// TIA Portal V15.1 export
// export: Created 2024-06-21T08:41:15.0924027Z, ExportSetting WithDefaults, DisplayName Totally Integrated Automation Portal, DisplayVersion V15.1 Update 5, DisplayName TIA Portal Openness, DisplayVersion V15.1 Update 5, DisplayName SINAMICS Startdrive Advanced, DisplayVersion V15.1, DisplayName G130, G150, S120, S150, SINAMICS MV, S210, DisplayVersion V15.1, DisplayName G110M, G120, G120C, G120D, G120P, DisplayVersion V15.1, DisplayName STEP 7 Professional, DisplayVersion V15.1 Update 5, DisplayName STEP 7 Safety, DisplayVersion V15.1, DisplayName WinCC Professional, DisplayVersion V15.1 Update 5, DisplayName SIMATIC Visualization Architect, DisplayVersion V15.1
FUNCTION_BLOCK "LGBChain2W1S-MoviFitFCPN"   // FB6710, FBD
TITLE = LGBChain2W1S-C / LGBChain2W1S-MoviFitFCPN
{ S7_Optimized_Access := 'TRUE' }
VERSION : 0.1
// stored: AutoNumber false, IsIECCheckEnabled false, IsRetainMemResEnabled false, MemoryReserve 100, SetENOAutomatically False, UDAEnableTagReadback false
   VAR_INPUT
      I_ExitDet { ExternalAccessible := 'False'; ExternalVisible := 'False'; ExternalWritable := 'False'} : Bool;   // Stop Detection set
      I_EntranceDet { ExternalAccessible := 'False'; ExternalVisible := 'False'; ExternalWritable := 'False'} : Bool;   // Stop Detection Reset
      I_StopDetPrev { ExternalAccessible := 'False'; ExternalVisible := 'False'; ExternalWritable := 'False'} : Bool;   // Stop Detection previous conveyor
      I_SlipControlDet { ExternalAccessible := 'False'; ExternalVisible := 'False'; ExternalWritable := 'False'} : Bool;   // Slack Chain detection
      I_TrfInSetBegin { ExternalAccessible := 'False'; ExternalVisible := 'False'; ExternalWritable := 'False'} : Bool;   // Load Begin: condition to start transfer IN set
      I_TrfInSetIntlkOk { ExternalAccessible := 'False'; ExternalVisible := 'False'; ExternalWritable := 'False'} : Bool;   // Transfer IN Interlock Set OK
      I_TrfOutSetBegin { ExternalAccessible := 'False'; ExternalVisible := 'False'; ExternalWritable := 'False'} : Bool;   // Unload Begin: condition to start transfer OUT set
      I_TrfOutSetIntlkOk { ExternalAccessible := 'False'; ExternalVisible := 'False'; ExternalWritable := 'False'} : Bool;   // Transfer Out Interlock Set OK
      I_TrfInSetRdyDlv { ExternalAccessible := 'False'; ExternalVisible := 'False'; ExternalWritable := 'False'} : Bool;   // Ready to deliver: Signal from previous object set
      I_TrfInSetTM { ExternalAccessible := 'False'; ExternalVisible := 'False'; ExternalWritable := 'False'} : Bool;   // Transfer busy signal from previous equipement set
      I_TrfOutSetRdyRcv { ExternalAccessible := 'False'; ExternalVisible := 'False'; ExternalWritable := 'False'} : Bool;   // Ready to Receive: Signal from next object set
      I_TrfOutSetArrived { ExternalAccessible := 'False'; ExternalVisible := 'False'; ExternalWritable := 'False'} : Bool;   // Body Arrived: Signal from next object Set
      I_PBSet { ExternalAccessible := 'False'; ExternalVisible := 'False'; ExternalWritable := 'False'} : Bool;   // Push button for manual movement (on local panel) set
      I_PBReset { ExternalAccessible := 'False'; ExternalVisible := 'False'; ExternalWritable := 'False'} : Bool;   // Push button for manual movement (on local panel) Reset
      I_ManInfeedAllowedSet { ExternalAccessible := 'False'; ExternalVisible := 'False'; ExternalWritable := 'False'} : Bool;   // Manual Infeed Allowed Set (without PushButton)
      I_ManInfeedAllowedRes { ExternalAccessible := 'False'; ExternalVisible := 'False'; ExternalWritable := 'False'} : Bool;   // Manual Infeed Allowed Reset (without PushButton)
      I_MotorProtection { ExternalAccessible := 'False'; ExternalVisible := 'False'; ExternalWritable := 'False'} : Bool;   // Motorprotection
      I_ReleaseBrake { ExternalAccessible := 'False'; ExternalVisible := 'False'; ExternalWritable := 'False'} : Bool;   // Release brake
      I_SafetyOk { ExternalAccessible := 'False'; ExternalVisible := 'False'; ExternalWritable := 'False'} : Bool;   // Safety Ok
      I_MotionStopOk { ExternalAccessible := 'False'; ExternalVisible := 'False'; ExternalWritable := 'False'} : Bool;   // Safety Ok / The motion stop is Ok
      I_ProductionStop { ExternalAccessible := 'False'; ExternalVisible := 'False'; ExternalWritable := 'False'} : Bool;   // Production Stop
      I_ExtStartConveyor { ExternalAccessible := 'False'; ExternalVisible := 'False'; ExternalWritable := 'False'} : Bool;   // External Start Conveyor
      I_ChainEmptyTime { ExternalAccessible := 'False'; ExternalVisible := 'False'; ExternalWritable := 'False'} : DInt;   // Time to empty Chain (Msec)
      I_Speed { ExternalAccessible := 'False'; ExternalVisible := 'False'; ExternalWritable := 'False'} : Real;   // High speed Value (set-up %) / Speed Value (set-up %)
      I_SafetyStatusWord { ExternalAccessible := 'False'; ExternalVisible := 'False'; ExternalWritable := 'False'} : Word;   // Safety Status
      I_SafetyControlWord { ExternalAccessible := 'False'; ExternalVisible := 'False'; ExternalWritable := 'False'} : Word;   // Safety Control Word
   END_VAR
   VAR_OUTPUT
      O_ReleaseBrake { ExternalAccessible := 'False'; ExternalVisible := 'False'; ExternalWritable := 'False'} : Bool;   // Release the brake of the Motor
      O_Active { ExternalAccessible := 'False'; ExternalVisible := 'False'; ExternalWritable := 'False'} : Bool;   // Chain is Active
      O_TrfInSetRdyRcv { ExternalAccessible := 'False'; ExternalVisible := 'False'; ExternalWritable := 'False'} : Bool;   // Ready to Receive: Signal to previous object set
      O_TrfInSetArrived { ExternalAccessible := 'False'; ExternalVisible := 'False'; ExternalWritable := 'False'} : Bool;   // Body Arrived: Signal to previous object Set
      O_TrfOutSetRdyDlv { ExternalAccessible := 'False'; ExternalVisible := 'False'; ExternalWritable := 'False'} : Bool;   // Ready to Deliver: Signal to next object set
      O_TrfOutSetTM { ExternalAccessible := 'False'; ExternalVisible := 'False'; ExternalWritable := 'False'} : Bool;   // Transfer: Signal to next object set
      O_TrfInSetActive { ExternalAccessible := 'False'; ExternalVisible := 'False'; ExternalWritable := 'False'} : Bool;   // Transfer in set active
      O_TrfInSetFinished { ExternalAccessible := 'False'; ExternalVisible := 'False'; ExternalWritable := 'False'} : Bool;   // Transfer in set finished
      O_TrfOutSetActive { ExternalAccessible := 'False'; ExternalVisible := 'False'; ExternalWritable := 'False'} : Bool;   // Transfer out set active
      O_TrfOutSetFinished { ExternalAccessible := 'False'; ExternalVisible := 'False'; ExternalWritable := 'False'} : Bool;   // Transfer out set finished
      O_LedRoller { ExternalAccessible := 'False'; ExternalVisible := 'False'; ExternalWritable := 'False'} : Bool;   // Led of Chain
      O_AlarmABCondition { ExternalAccessible := 'False'; ExternalVisible := 'False'; ExternalWritable := 'False'} : Bool;   // Alarm AB Condition
      O_AlarmA { ExternalAccessible := 'False'; ExternalVisible := 'False'; ExternalWritable := 'False'} : Bool;   // Alarm A
      O_AlarmB { ExternalAccessible := 'False'; ExternalVisible := 'False'; ExternalWritable := 'False'} : Bool;   // Alarm B
      O_AlarmC { ExternalAccessible := 'False'; ExternalVisible := 'False'; ExternalWritable := 'False'} : Bool;   // Alarm C
      O_AlarmD { ExternalAccessible := 'False'; ExternalVisible := 'False'; ExternalWritable := 'False'} : Bool;   // Alarm D
      O_Occupied { ExternalAccessible := 'False'; ExternalVisible := 'False'; ExternalWritable := 'False'} : Bool;   // Chain Occupied
      H_AlarmDWord { ExternalAccessible := 'False'; ExternalVisible := 'False'; ExternalWritable := 'False'} : DWord;   // HMI Animation
   END_VAR
   VAR_IN_OUT
      IO_Modes : "Modes";   // Modes
      H_HMI : "H_HMI";   // Animation
      "H_GBChain2W1S-MoviFitFCPN" : "H_GBChain2W1S-MoviFitFCPN";   // Animation
      C_Config : "RollerConvMoviFitFCPNConfig";   // Config
   END_VAR
   VAR
      H_FncSelInHMI { ExternalAccessible := 'False'; ExternalVisible := 'False'; ExternalWritable := 'False'} : Bool;
      _SlipControl { ExternalAccessible := 'False'; ExternalVisible := 'False'; ExternalWritable := 'False'} : "L1AlarmMultiIn";   // FB
      _InitSlipControlCnt { ExternalAccessible := 'False'; ExternalVisible := 'False'; ExternalWritable := 'False'} : "LChangeOfState";   // FB
      AB_SlipControlAlm { ExternalAccessible := 'False'; ExternalVisible := 'False'; ExternalWritable := 'False'} : Bool;   // Alarm Slack Chain
      AC_TrfOutSetOverTime { ExternalAccessible := 'False'; ExternalVisible := 'False'; ExternalWritable := 'False'} : Bool;   // Timeout Transport Out Set
      AD_TrfOutSetInterlock { ExternalAccessible := 'False'; ExternalVisible := 'False'; ExternalWritable := 'False'} : Bool;   // Interlock Not Ok Transport Out Set
      AD_TrfInSetInterlock { ExternalAccessible := 'False'; ExternalVisible := 'False'; ExternalWritable := 'False'} : Bool;   // Interlock Not Ok Transport In Set
      AA_MotorProtector { ExternalAccessible := 'False'; ExternalVisible := 'False'; ExternalWritable := 'False'} : Bool;   // Motor Protection Tripped / Motorprotection Tripped
      AA_SafetySwitch { ExternalAccessible := 'False'; ExternalVisible := 'False'; ExternalWritable := 'False'} : Bool;   // Safety Switch Not Ok
      AB_STO { ExternalAccessible := 'False'; ExternalVisible := 'False'; ExternalWritable := 'False'} : Bool;   // Safety Switch Not Ok / Safety output to drive is active but no response from drive that the safety is ok
      AD_Warning { ExternalAccessible := 'False'; ExternalVisible := 'False'; ExternalWritable := 'False'} : Bool;   // Frequency Control
      AA_NoBusControl { ExternalAccessible := 'False'; ExternalVisible := 'False'; ExternalWritable := 'False'} : Bool;   // Frequency Control / Bus control inactive / Frekvensstyrning
      AB_Alarm { ExternalAccessible := 'False'; ExternalVisible := 'False'; ExternalWritable := 'False'} : Bool;   // Frequency Control
      AD_MotionStop { ExternalAccessible := 'False'; ExternalVisible := 'False'; ExternalWritable := 'False'} : Bool;   // Motion Stop
      AC_ConfigCalibrationAlm { ExternalAccessible := 'False'; ExternalVisible := 'False'; ExternalWritable := 'False'} : Bool;   // The Config values for Alarm Transfer time must be ALL zero or ALL different from zero
      AD_CalibrationSetWarn { ExternalAccessible := 'False'; ExternalVisible := 'False'; ExternalWritable := 'False'} : Bool;   // No High speed selected so Calibration is not possible for SET direction
      AC_ConfigRampAlm { ExternalAccessible := 'False'; ExternalVisible := 'False'; ExternalWritable := 'False'} : Bool;   // The config value for the ramp is not correct, must be zero or the config values for the calculation of the ramp must be ALL zero
      AC_ConfigRampCalcAlm { ExternalAccessible := 'False'; ExternalVisible := 'False'; ExternalWritable := 'False'} : Bool;   // The config values for the calculation of the ramp must be ALL different from zero
      PODataNotEnabled { ExternalAccessible := 'False'; ExternalVisible := 'False'; ExternalWritable := 'False'} : Bool;   // Bus control inactive
      SafetyOk { ExternalAccessible := 'False'; ExternalVisible := 'False'; ExternalWritable := 'False'} : Bool;   // Safety Ok
      SlipControlCond { ExternalAccessible := 'False'; ExternalVisible := 'False'; ExternalWritable := 'False'} : Bool;   // Alarm Slack Chain
      MotorLoopActive { ExternalAccessible := 'False'; ExternalVisible := 'False'; ExternalWritable := 'False'} : Bool;   // Motor Loop Active
      TrfInfeedHoldSet { ExternalAccessible := 'False'; ExternalVisible := 'False'; ExternalWritable := 'False'} : Bool;   // Transfer infeed hold set direction
      TrfOutSetCmd { ExternalAccessible := 'False'; ExternalVisible := 'False'; ExternalWritable := 'False'} : Bool;   // Command after Interlock to Motor set
      TrfOutfeedHoldSet { ExternalAccessible := 'False'; ExternalVisible := 'False'; ExternalWritable := 'False'} : Bool;   // Transfer outfeed hold set direction
      TrfInSetCmd { ExternalAccessible := 'False'; ExternalVisible := 'False'; ExternalWritable := 'False'} : Bool;   // Command after Interlock to Motor set
      MotorCmdSet { ExternalAccessible := 'False'; ExternalVisible := 'False'; ExternalWritable := 'False'} : Bool;   // Command to Motorloop High Speed Set
      MotorCmdRes { ExternalAccessible := 'False'; ExternalVisible := 'False'; ExternalWritable := 'False'} : Bool;   // Command to Motorloop High Speed Reset
      TrfInSetActive { ExternalAccessible := 'False'; ExternalVisible := 'False'; ExternalWritable := 'False'} : Bool;   // Load: Active (set)
      TrfOutSetActive { ExternalAccessible := 'False'; ExternalVisible := 'False'; ExternalWritable := 'False'} : Bool;   // Unload: active (set)
      TrfOutSetFinished { ExternalAccessible := 'False'; ExternalVisible := 'False'; ExternalWritable := 'False'} : Bool;   // Unload: finished (set)
      AlarmA { ExternalAccessible := 'False'; ExternalVisible := 'False'; ExternalWritable := 'False'} : Bool;   // Alarm A
      AlarmB { ExternalAccessible := 'False'; ExternalVisible := 'False'; ExternalWritable := 'False'} : Bool;   // Alarm B
      AlarmC { ExternalAccessible := 'False'; ExternalVisible := 'False'; ExternalWritable := 'False'} : Bool;   // Alarm C
      AlarmD { ExternalAccessible := 'False'; ExternalVisible := 'False'; ExternalWritable := 'False'} : Bool;   // Alarm D
      TrfOutSetRdyDlv { ExternalAccessible := 'False'; ExternalVisible := 'False'; ExternalWritable := 'False'} : Bool;   // Ready to Deliver: Signal to next object set
      TrfOutSetTM { ExternalAccessible := 'False'; ExternalVisible := 'False'; ExternalWritable := 'False'} : Bool;   // Transfer : Signal transfer memory to next object set
      TrfInSetTrfOutSetTM { ExternalAccessible := 'False'; ExternalVisible := 'False'; ExternalWritable := 'False'} : Bool;   // Transfer memory set
      TrfInSetRdyRcv { ExternalAccessible := 'False'; ExternalVisible := 'False'; ExternalWritable := 'False'} : Bool;   // Ready to Receive: Signal to previous object set
      TrfInSetArrived { ExternalAccessible := 'False'; ExternalVisible := 'False'; ExternalWritable := 'False'} : Bool;   // Body Arrived: Signal to previous object Set
      TrfInSetFinished { ExternalAccessible := 'False'; ExternalVisible := 'False'; ExternalWritable := 'False'} : Bool;   // Body Arrived: Signal to TrfOut module set (Reset TrfOutCmd)
      StopTrfOutSetCmd { ExternalAccessible := 'False'; ExternalVisible := 'False'; ExternalWritable := 'False'} : Bool;   // Body Arrived: Signal to previous object Set
      MotorLoopAlmCond { ExternalAccessible := 'False'; ExternalVisible := 'False'; ExternalWritable := 'False'} : Bool;   // Motor loop Alarm condition
      TrfOutSetAlmCond { ExternalAccessible := 'False'; ExternalVisible := 'False'; ExternalWritable := 'False'} : Bool;   // TrfOut set Alarm condition
      ChainStop { ExternalAccessible := 'False'; ExternalVisible := 'False'; ExternalWritable := 'False'} : Bool;   // Chain stop Productions Stop
      DlvSaturation { ExternalAccessible := 'False'; ExternalVisible := 'False'; ExternalWritable := 'False'} : Bool;   // Saturation for the diliver tranfer
      AlarmABCondition { ExternalAccessible := 'False'; ExternalVisible := 'False'; ExternalWritable := 'False'} : Bool;   // Alarm AB Condition
   END_VAR
   VAR RETAIN
      ChainEmpty { ExternalAccessible := 'False'; ExternalVisible := 'False'; ExternalWritable := 'False'} : Bool;   // Chain is Empty
   END_VAR
   VAR
      ChainEmptyTime { ExternalAccessible := 'False'; ExternalVisible := 'False'; ExternalWritable := 'False'} : DInt;   // Time to empty Chain (Msec)
      SlipControlPulseCount { ExternalAccessible := 'False'; ExternalVisible := 'False'; ExternalWritable := 'False'} : DInt;   // Temp
      SlipControlPosEdge1 { ExternalAccessible := 'False'; ExternalVisible := 'False'; ExternalWritable := 'False'} : Bool;   // Pos Edge
      SlipControlPosEdge2 { ExternalAccessible := 'False'; ExternalVisible := 'False'; ExternalWritable := 'False'} : Bool;   // Pos Edge
      InitSlipControlCounter { ExternalAccessible := 'False'; ExternalVisible := 'False'; ExternalWritable := 'False'} : Bool;   // Init
      ReleaseBrake { ExternalAccessible := 'False'; ExternalVisible := 'False'; ExternalWritable := 'False'} : Bool;   // Release brake
      ReadyForOperation { ExternalAccessible := 'False'; ExternalVisible := 'False'; ExternalWritable := 'False'} : Bool;   // Ready for operation
      _LTrfInSet { ExternalAccessible := 'False'; ExternalVisible := 'False'; ExternalWritable := 'False'} : "LGBTrfIn";   // FB
      _LTrfOutSet { ExternalAccessible := 'False'; ExternalVisible := 'False'; ExternalWritable := 'False'} : "LGBTrfOut";   // FB
      _Motor { ExternalAccessible := 'False'; ExternalVisible := 'False'; ExternalWritable := 'False'} : "LGBMotor2W2S-MoviFitFCPN";
      _ChainSlipControl { ExternalAccessible := 'False'; ExternalVisible := 'False'; ExternalWritable := 'False'} : "L1AlarmMultiIn";
      _ChainEmptyTimer { ExternalAccessible := 'False'; ExternalVisible := 'False'; ExternalWritable := 'False'} : TON_TIME;
   END_VAR
   VAR_TEMP
      H_HMITrfInSet : "H_HMI";   // Temp
      H_HMITrfOutSet : "H_HMI";   // Temp
      H_HMIMotor : "H_HMI";   // Temp
   END_VAR
   VAR_TEMP   // added for the SCL form of the ladder/FBD networks
      _w1 : Bool;
      _w2 : Bool;
      _w3 : Bool;
      _w4 : Bool;
   END_VAR
BEGIN

NETWORK
TITLE = **** 1 - Inputs **** Init Slip Control Set Direction
// Init Belt Control Set And Reset Direction
      CALL  #_InitSlipControlCnt
      ( I_In     := #I_SlipControlDet,
        O_OutPut := #InitSlipControlCounter
      );
      NOP   0;

      A(;
      O     #InitSlipControlCounter;
      O;
      A     #IO_Modes.LMode.ManualMode;
      A     #IO_Modes.LMode.AlarmResetPB;
      );
      JCN   NCSet;
      L     0;
      T     #SlipControlPulseCount;
NCSet:NOP   0;


REGION Network 2: **** 1 - Inputs **** Safety Ok
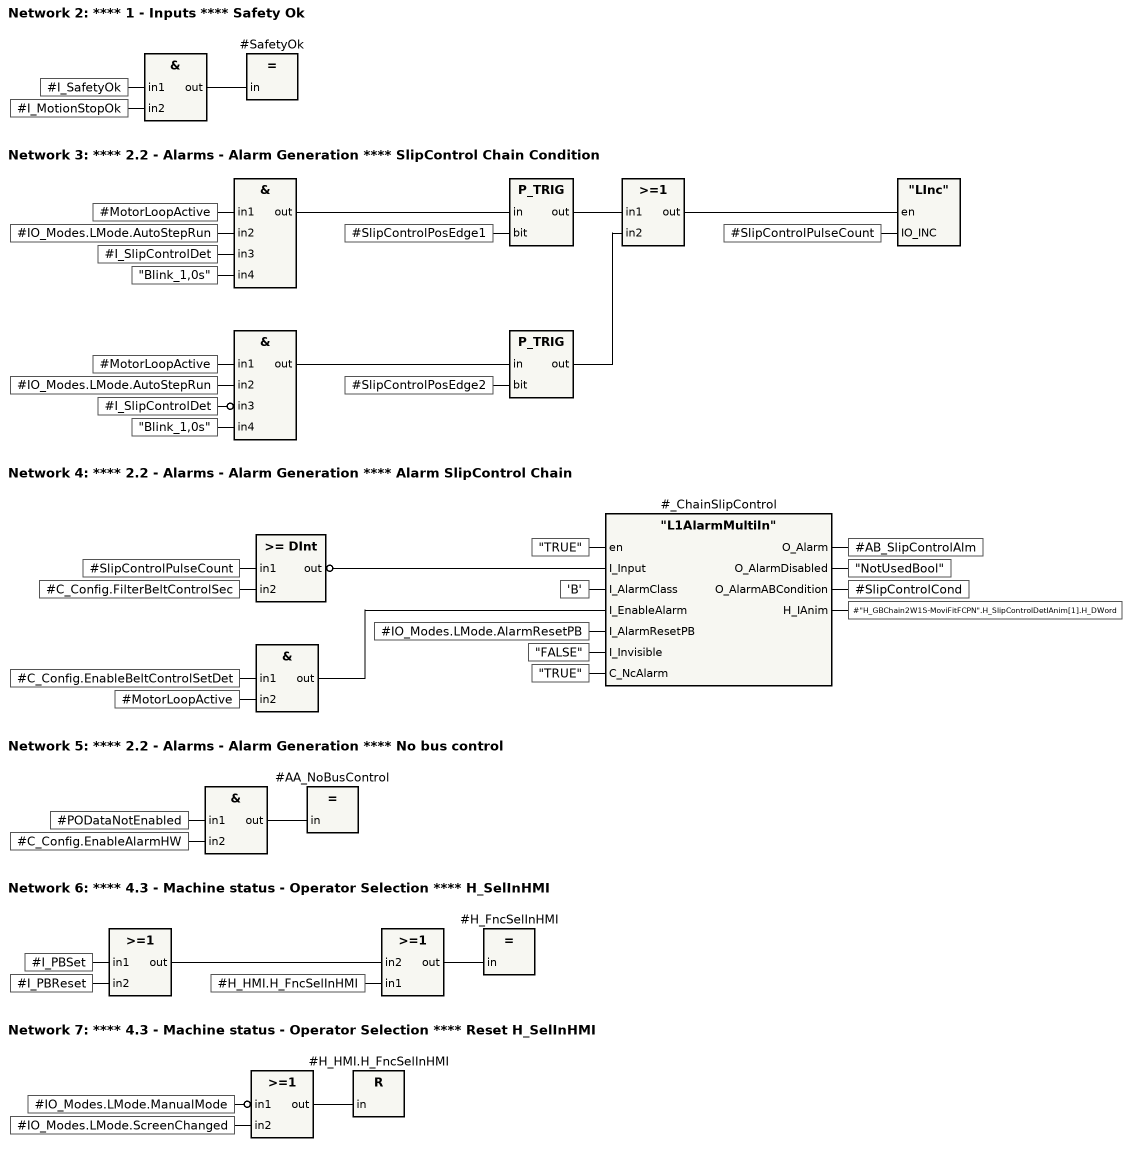
   #SafetyOk := #I_SafetyOk AND #I_MotionStopOk;
END_REGION

REGION Network 3: **** 2.2 - Alarms - Alarm Generation **** SlipControl Chain Condition
   // Belt Control CrossConv Set Condition
   #_w1 := #MotorLoopActive AND #IO_Modes.LMode.AutoStepRun AND #I_SlipControlDet AND "Blink_1,0s";
   #_w2 := #_w1 AND NOT #SlipControlPosEdge1;   // rising edge
   #SlipControlPosEdge1 := #_w1;
   #_w3 := #MotorLoopActive AND #IO_Modes.LMode.AutoStepRun AND NOT #I_SlipControlDet AND "Blink_1,0s";
   #_w4 := #_w3 AND NOT #SlipControlPosEdge2;   // rising edge
   #SlipControlPosEdge2 := #_w3;
   IF #_w2 OR #_w4 THEN "LInc"(IO_INC := #SlipControlPulseCount); END_IF;
END_REGION

REGION Network 4: **** 2.2 - Alarms - Alarm Generation **** Alarm SlipControl Chain
   // Alarm Slack Chain
   IF "TRUE" THEN
       #_ChainSlipControl(I_Input := NOT (#SlipControlPulseCount >= #C_Config.FilterBeltControlSec),   // "L1AlarmMultiIn"
                          I_AlarmClass := 'B',
                          I_EnableAlarm := #C_Config.EnableBeltControlSetDet AND #MotorLoopActive,
                          I_AlarmResetPB := #IO_Modes.LMode.AlarmResetPB,
                          I_Invisible := "FALSE",
                          C_NcAlarm := "TRUE",
                          O_Alarm => #AB_SlipControlAlm,
                          O_AlarmDisabled => "NotUsedBool",
                          O_AlarmABCondition => #SlipControlCond,
                          H_IAnim => #"H_GBChain2W1S-MoviFitFCPN".H_SlipControlDetIAnim[1].H_DWord);
   END_IF;
END_REGION

REGION Network 5: **** 2.2 - Alarms - Alarm Generation **** No bus control
   #AA_NoBusControl := #PODataNotEnabled AND #C_Config.EnableAlarmHW;
END_REGION

REGION Network 6: **** 4.3 - Machine status - Operator Selection **** H_SelInHMI
   #H_FncSelInHMI := #I_PBSet OR #I_PBReset OR #H_HMI.H_FncSelInHMI;
END_REGION

REGION Network 7: **** 4.3 - Machine status - Operator Selection **** Reset H_SelInHMI
   // Reset H_SelInHMI
   IF NOT #IO_Modes.LMode.ManualMode OR #IO_Modes.LMode.ScreenChanged THEN
       #H_HMI.H_FncSelInHMI := FALSE;
   END_IF;
END_REGION

REGION Network 8: **** 4.4 - Machine status - Calculated **** Chain is empty
   // Chain is empty when chain is running and no detection is activated during the preset time
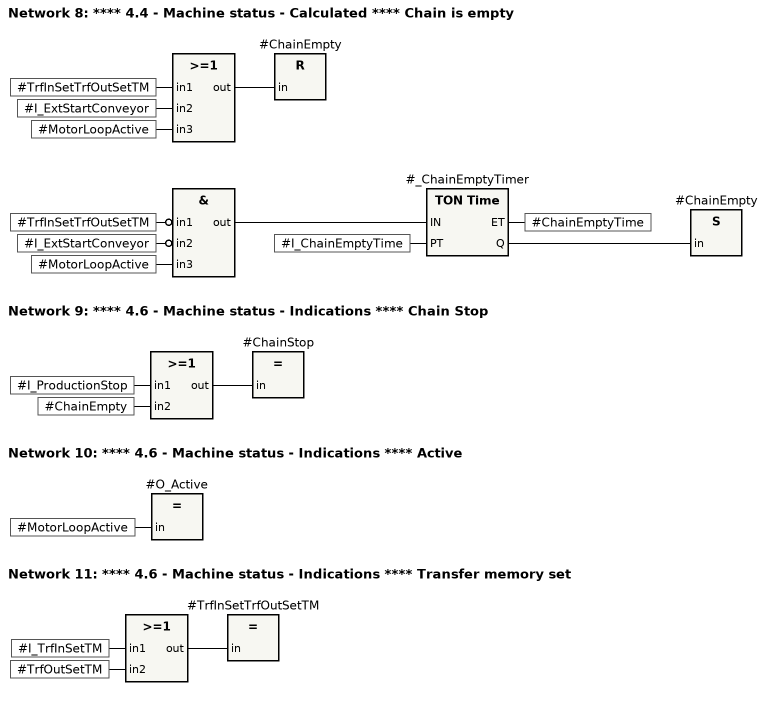
   IF #TrfInSetTrfOutSetTM OR #I_ExtStartConveyor OR #MotorLoopActive THEN #ChainEmpty := FALSE; END_IF;
   #_ChainEmptyTimer(IN := NOT #TrfInSetTrfOutSetTM AND NOT #I_ExtStartConveyor AND #MotorLoopActive,   // TON
                     PT := #I_ChainEmptyTime,
                     ET => #ChainEmptyTime);
   IF #_ChainEmptyTimer.Q THEN #ChainEmpty := TRUE; END_IF;
END_REGION

REGION Network 9: **** 4.6 - Machine status - Indications **** Chain Stop
   #ChainStop := #I_ProductionStop OR #ChainEmpty;
END_REGION

REGION Network 10: **** 4.6 - Machine status - Indications **** Active
   // Active
   #O_Active := #MotorLoopActive;
END_REGION

REGION Network 11: **** 4.6 - Machine status - Indications **** Transfer memory set
   // Transfer memory set
   #TrfInSetTrfOutSetTM := #I_TrfInSetTM OR #TrfOutSetTM;
END_REGION

REGION Network 12: **** 4.6 - Machine Status - Indication **** Entrance Det
   // Entrance Det
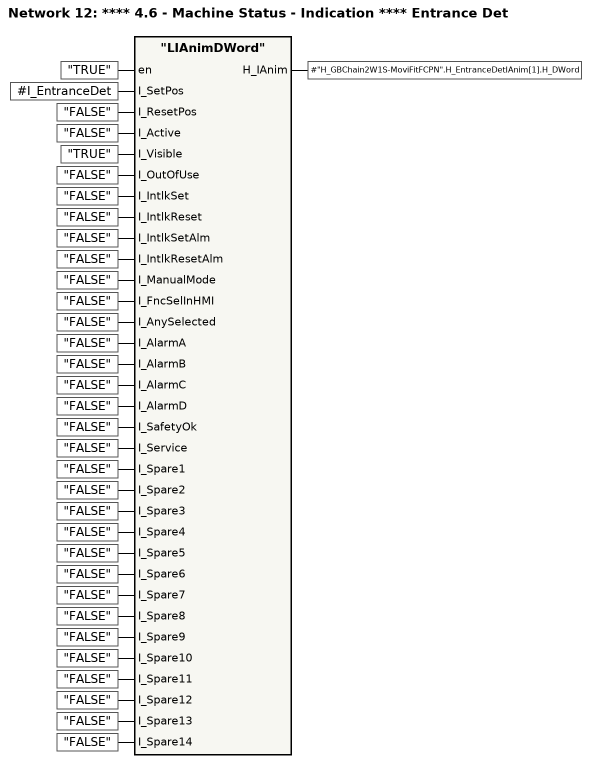
   IF "TRUE" THEN
       "LIAnimDWord"(I_SetPos := #I_EntranceDet,
                     I_ResetPos := "FALSE",
                     I_Active := "FALSE",
                     I_Visible := "TRUE",
                     I_OutOfUse := "FALSE",
                     I_IntlkSet := "FALSE",
                     I_IntlkReset := "FALSE",
                     I_IntlkSetAlm := "FALSE",
                     I_IntlkResetAlm := "FALSE",
                     I_ManualMode := "FALSE",
                     I_FncSelInHMI := "FALSE",
                     I_AnySelected := "FALSE",
                     I_AlarmA := "FALSE",
                     I_AlarmB := "FALSE",
                     I_AlarmC := "FALSE",
                     I_AlarmD := "FALSE",
                     I_SafetyOk := "FALSE",
                     I_Service := "FALSE",
                     I_Spare1 := "FALSE",
                     I_Spare2 := "FALSE",
                     I_Spare3 := "FALSE",
                     I_Spare4 := "FALSE",
                     I_Spare5 := "FALSE",
                     I_Spare6 := "FALSE",
                     I_Spare7 := "FALSE",
                     I_Spare8 := "FALSE",
                     I_Spare9 := "FALSE",
                     I_Spare10 := "FALSE",
                     I_Spare11 := "FALSE",
                     I_Spare12 := "FALSE",
                     I_Spare13 := "FALSE",
                     I_Spare14 := "FALSE",
                     H_IAnim => #"H_GBChain2W1S-MoviFitFCPN".H_EntranceDetIAnim[1].H_DWord);
   END_IF;
END_REGION

REGION Network 13: **** 4.6 - Machine Status - Indication **** Exit Det
   // Exit Det
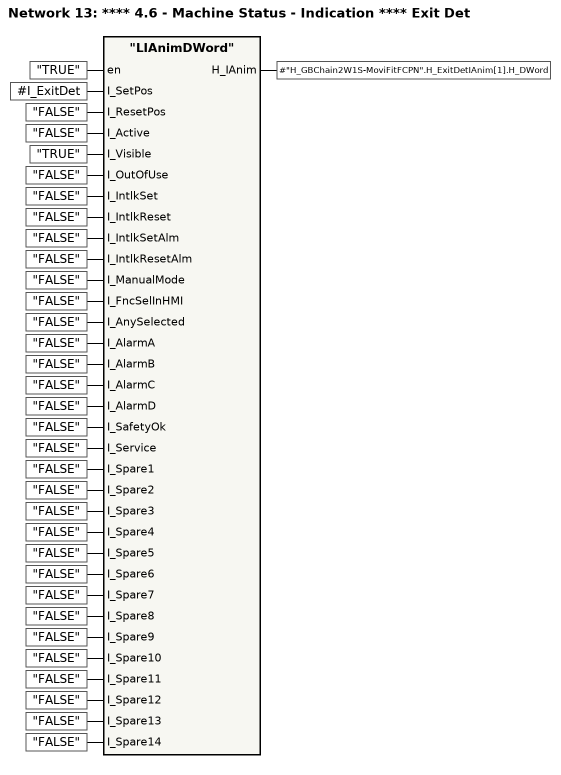
   IF "TRUE" THEN
       "LIAnimDWord"(I_SetPos := #I_ExitDet,
                     I_ResetPos := "FALSE",
                     I_Active := "FALSE",
                     I_Visible := "TRUE",
                     I_OutOfUse := "FALSE",
                     I_IntlkSet := "FALSE",
                     I_IntlkReset := "FALSE",
                     I_IntlkSetAlm := "FALSE",
                     I_IntlkResetAlm := "FALSE",
                     I_ManualMode := "FALSE",
                     I_FncSelInHMI := "FALSE",
                     I_AnySelected := "FALSE",
                     I_AlarmA := "FALSE",
                     I_AlarmB := "FALSE",
                     I_AlarmC := "FALSE",
                     I_AlarmD := "FALSE",
                     I_SafetyOk := "FALSE",
                     I_Service := "FALSE",
                     I_Spare1 := "FALSE",
                     I_Spare2 := "FALSE",
                     I_Spare3 := "FALSE",
                     I_Spare4 := "FALSE",
                     I_Spare5 := "FALSE",
                     I_Spare6 := "FALSE",
                     I_Spare7 := "FALSE",
                     I_Spare8 := "FALSE",
                     I_Spare9 := "FALSE",
                     I_Spare10 := "FALSE",
                     I_Spare11 := "FALSE",
                     I_Spare12 := "FALSE",
                     I_Spare13 := "FALSE",
                     I_Spare14 := "FALSE",
                     H_IAnim => #"H_GBChain2W1S-MoviFitFCPN".H_ExitDetIAnim[1].H_DWord);
   END_IF;
END_REGION

REGION Network 14: **** 4.6 - Machine Status - Indication **** Icon Animation
   // Icon Animation
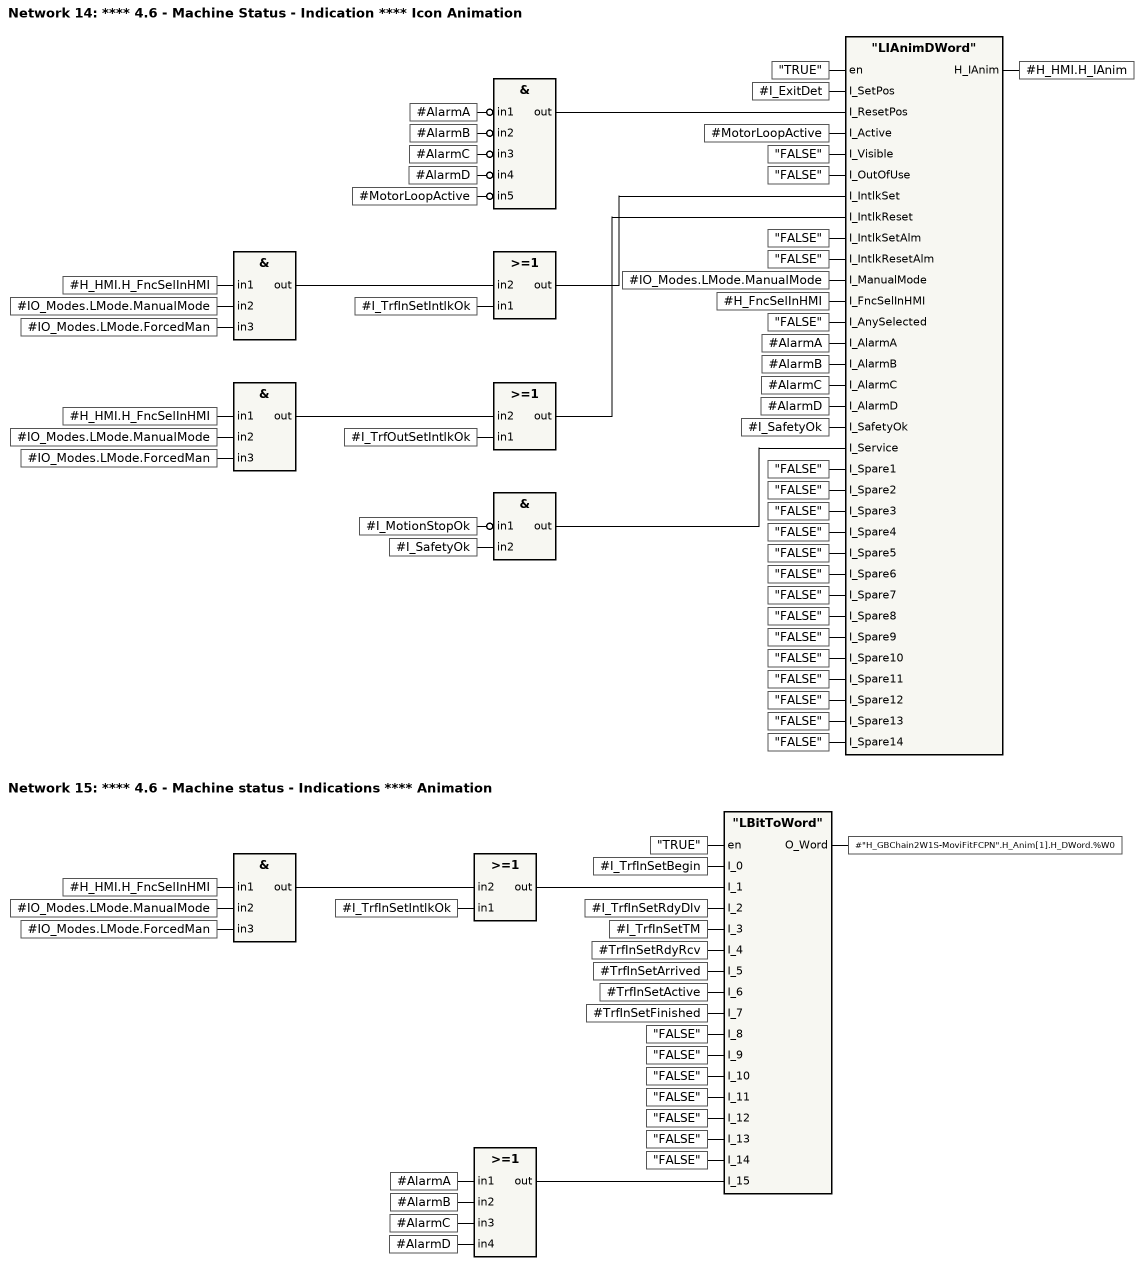
   IF "TRUE" THEN
       "LIAnimDWord"(I_SetPos := #I_ExitDet,
                     I_ResetPos := NOT #AlarmA AND NOT #AlarmB AND NOT #AlarmC AND NOT #AlarmD AND NOT #MotorLoopActive,
                     I_Active := #MotorLoopActive,
                     I_Visible := "FALSE",
                     I_OutOfUse := "FALSE",
                     I_IntlkSet := (#H_HMI.H_FncSelInHMI AND #IO_Modes.LMode.ManualMode AND #IO_Modes.LMode.ForcedMan) OR #I_TrfInSetIntlkOk,
                     I_IntlkReset := (#H_HMI.H_FncSelInHMI AND #IO_Modes.LMode.ManualMode AND #IO_Modes.LMode.ForcedMan) OR #I_TrfOutSetIntlkOk,
                     I_IntlkSetAlm := "FALSE",
                     I_IntlkResetAlm := "FALSE",
                     I_ManualMode := #IO_Modes.LMode.ManualMode,
                     I_FncSelInHMI := #H_FncSelInHMI,
                     I_AnySelected := "FALSE",
                     I_AlarmA := #AlarmA,
                     I_AlarmB := #AlarmB,
                     I_AlarmC := #AlarmC,
                     I_AlarmD := #AlarmD,
                     I_SafetyOk := #I_SafetyOk,
                     I_Service := NOT #I_MotionStopOk AND #I_SafetyOk,
                     I_Spare1 := "FALSE",
                     I_Spare2 := "FALSE",
                     I_Spare3 := "FALSE",
                     I_Spare4 := "FALSE",
                     I_Spare5 := "FALSE",
                     I_Spare6 := "FALSE",
                     I_Spare7 := "FALSE",
                     I_Spare8 := "FALSE",
                     I_Spare9 := "FALSE",
                     I_Spare10 := "FALSE",
                     I_Spare11 := "FALSE",
                     I_Spare12 := "FALSE",
                     I_Spare13 := "FALSE",
                     I_Spare14 := "FALSE",
                     H_IAnim => #H_HMI.H_IAnim);
   END_IF;
END_REGION

REGION Network 15: **** 4.6 - Machine status - Indications **** Animation
   // Animation
   IF "TRUE" THEN
       "LBitToWord"(I_0 := #I_TrfInSetBegin,
                    I_1 := (#H_HMI.H_FncSelInHMI AND #IO_Modes.LMode.ManualMode AND #IO_Modes.LMode.ForcedMan) OR #I_TrfInSetIntlkOk,
                    I_2 := #I_TrfInSetRdyDlv,
                    I_3 := #I_TrfInSetTM,
                    I_4 := #TrfInSetRdyRcv,
                    I_5 := #TrfInSetArrived,
                    I_6 := #TrfInSetActive,
                    I_7 := #TrfInSetFinished,
                    I_8 := "FALSE",
                    I_9 := "FALSE",
                    I_10 := "FALSE",
                    I_11 := "FALSE",
                    I_12 := "FALSE",
                    I_13 := "FALSE",
                    I_14 := "FALSE",
                    I_15 := #AlarmA OR #AlarmB OR #AlarmC OR #AlarmD,
                    O_Word => #"H_GBChain2W1S-MoviFitFCPN".H_Anim[1].H_DWord.%W0);
   END_IF;
END_REGION

REGION Network 16: **** 4.6 - Machine status - Indications **** Animation
   // Animation
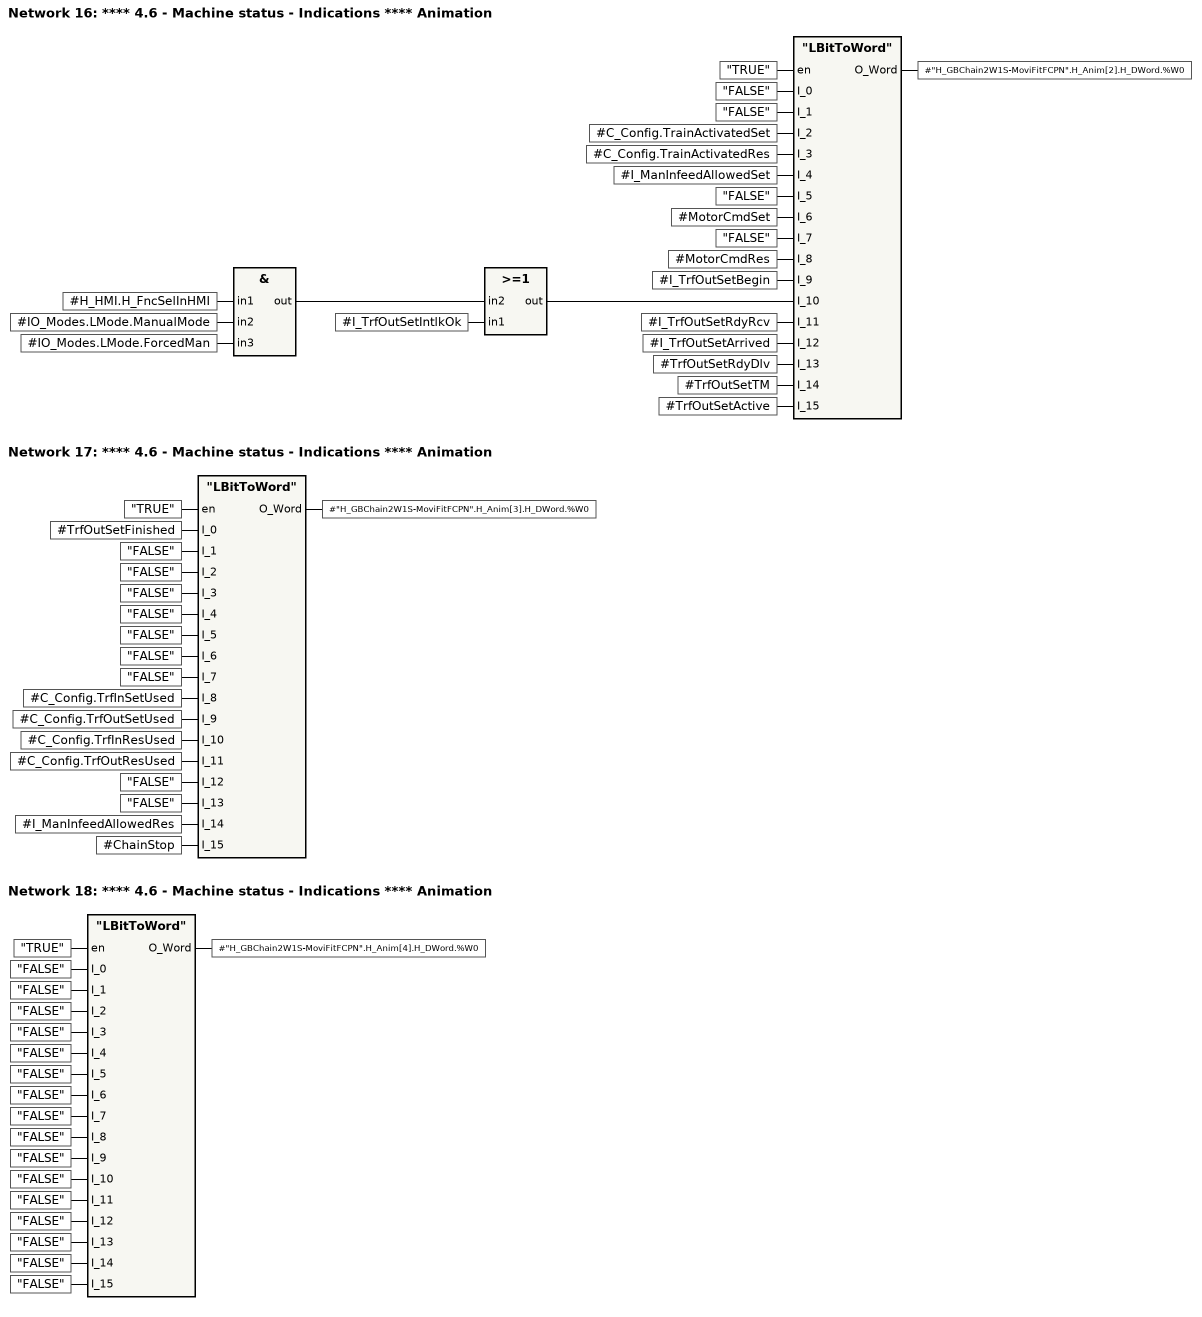
   IF "TRUE" THEN
       "LBitToWord"(I_0 := "FALSE",
                    I_1 := "FALSE",
                    I_2 := #C_Config.TrainActivatedSet,
                    I_3 := #C_Config.TrainActivatedRes,
                    I_4 := #I_ManInfeedAllowedSet,
                    I_5 := "FALSE",
                    I_6 := #MotorCmdSet,
                    I_7 := "FALSE",
                    I_8 := #MotorCmdRes,
                    I_9 := #I_TrfOutSetBegin,
                    I_10 := (#H_HMI.H_FncSelInHMI AND #IO_Modes.LMode.ManualMode AND #IO_Modes.LMode.ForcedMan) OR #I_TrfOutSetIntlkOk,
                    I_11 := #I_TrfOutSetRdyRcv,
                    I_12 := #I_TrfOutSetArrived,
                    I_13 := #TrfOutSetRdyDlv,
                    I_14 := #TrfOutSetTM,
                    I_15 := #TrfOutSetActive,
                    O_Word => #"H_GBChain2W1S-MoviFitFCPN".H_Anim[2].H_DWord.%W0);
   END_IF;
END_REGION

REGION Network 17: **** 4.6 - Machine status - Indications **** Animation
   // Animation
   IF "TRUE" THEN
       "LBitToWord"(I_0 := #TrfOutSetFinished,
                    I_1 := "FALSE",
                    I_2 := "FALSE",
                    I_3 := "FALSE",
                    I_4 := "FALSE",
                    I_5 := "FALSE",
                    I_6 := "FALSE",
                    I_7 := "FALSE",
                    I_8 := #C_Config.TrfInSetUsed,
                    I_9 := #C_Config.TrfOutSetUsed,
                    I_10 := #C_Config.TrfInResUsed,
                    I_11 := #C_Config.TrfOutResUsed,
                    I_12 := "FALSE",
                    I_13 := "FALSE",
                    I_14 := #I_ManInfeedAllowedRes,
                    I_15 := #ChainStop,
                    O_Word => #"H_GBChain2W1S-MoviFitFCPN".H_Anim[3].H_DWord.%W0);
   END_IF;
END_REGION

REGION Network 18: **** 4.6 - Machine status - Indications **** Animation
   // Animation
   IF "TRUE" THEN
       "LBitToWord"(I_0 := "FALSE",
                    I_1 := "FALSE",
                    I_2 := "FALSE",
                    I_3 := "FALSE",
                    I_4 := "FALSE",
                    I_5 := "FALSE",
                    I_6 := "FALSE",
                    I_7 := "FALSE",
                    I_8 := "FALSE",
                    I_9 := "FALSE",
                    I_10 := "FALSE",
                    I_11 := "FALSE",
                    I_12 := "FALSE",
                    I_13 := "FALSE",
                    I_14 := "FALSE",
                    I_15 := "FALSE",
                    O_Word => #"H_GBChain2W1S-MoviFitFCPN".H_Anim[4].H_DWord.%W0);
   END_IF;
END_REGION

REGION Network 19: **** 4.6 - Machine status - Indications **** Animation Time Chain Stop
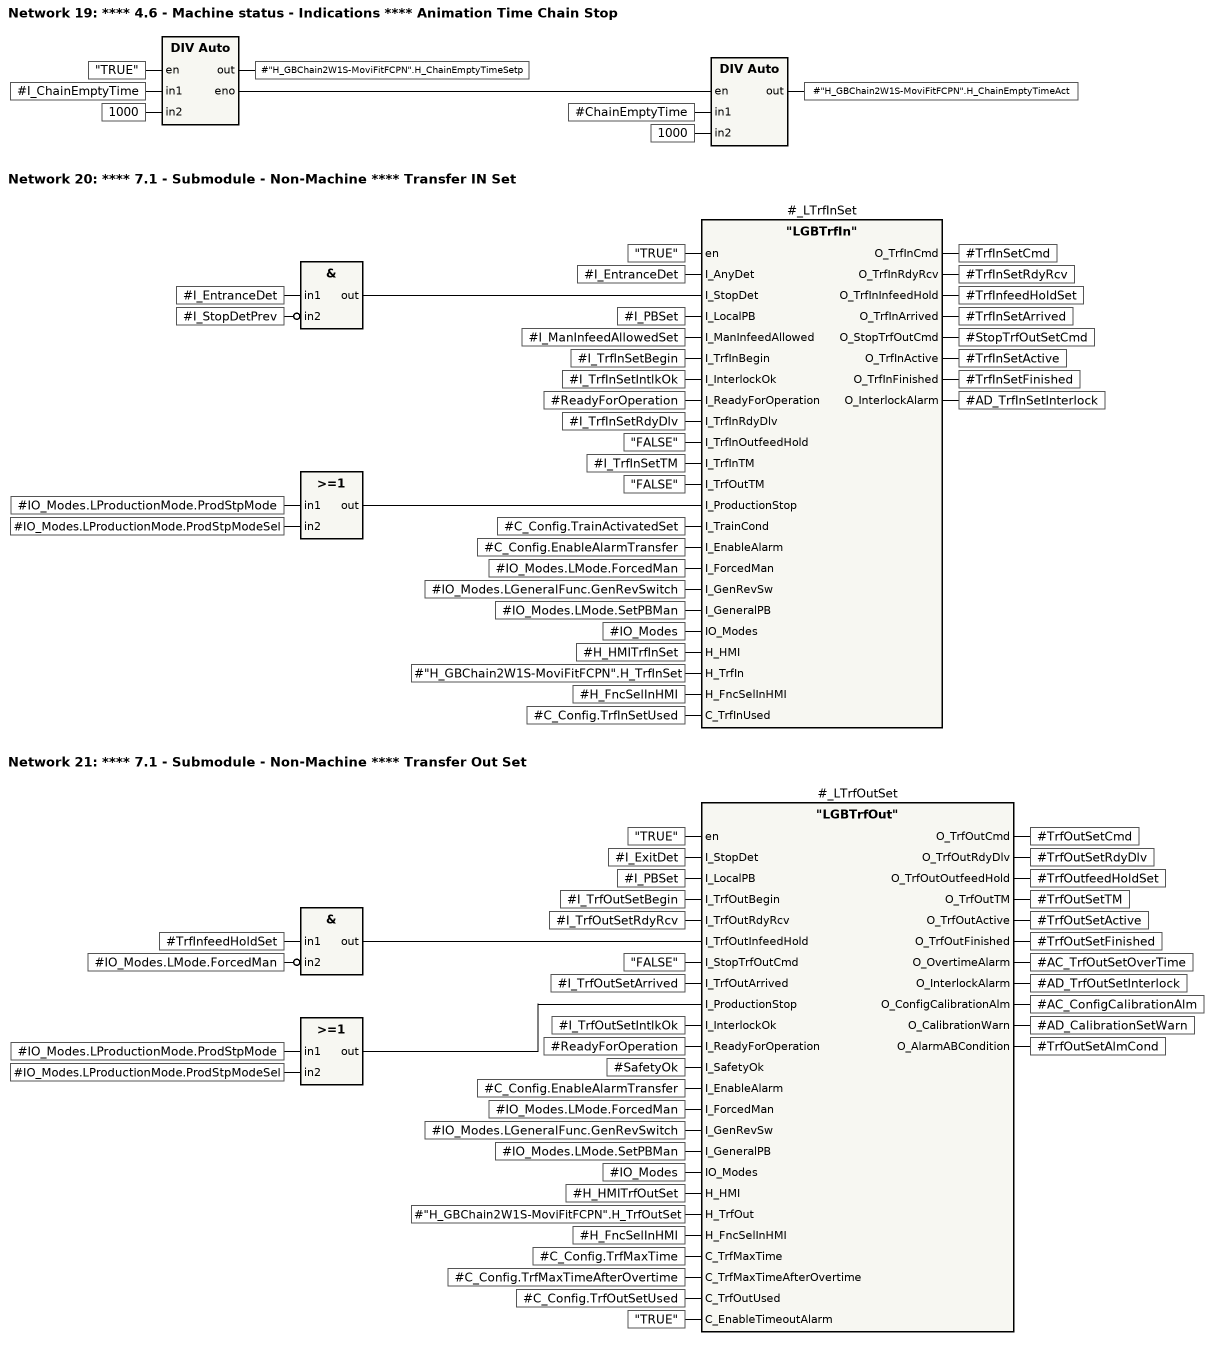
   IF "TRUE" THEN
       #"H_GBChain2W1S-MoviFitFCPN".H_ChainEmptyTimeSetp := #I_ChainEmptyTime / 1000;
       #"H_GBChain2W1S-MoviFitFCPN".H_ChainEmptyTimeAct := #ChainEmptyTime / 1000;
   END_IF;
END_REGION

REGION Network 20: **** 7.1 - Submodule - Non-Machine **** Transfer IN Set
   // Transfer IN Set
   IF "TRUE" THEN
       #_LTrfInSet(I_AnyDet := #I_EntranceDet,   // "LGBTrfIn"
                   I_StopDet := #I_EntranceDet AND NOT #I_StopDetPrev,
                   I_LocalPB := #I_PBSet,
                   I_ManInfeedAllowed := #I_ManInfeedAllowedSet,
                   I_TrfInBegin := #I_TrfInSetBegin,
                   I_InterlockOk := #I_TrfInSetIntlkOk,
                   I_ReadyForOperation := #ReadyForOperation,
                   I_TrfInRdyDlv := #I_TrfInSetRdyDlv,
                   I_TrfInOutfeedHold := "FALSE",
                   I_TrfInTM := #I_TrfInSetTM,
                   I_TrfOutTM := "FALSE",
                   I_ProductionStop := #IO_Modes.LProductionMode.ProdStpMode OR #IO_Modes.LProductionMode.ProdStpModeSel,
                   I_TrainCond := #C_Config.TrainActivatedSet,
                   I_EnableAlarm := #C_Config.EnableAlarmTransfer,
                   I_ForcedMan := #IO_Modes.LMode.ForcedMan,
                   I_GenRevSw := #IO_Modes.LGeneralFunc.GenRevSwitch,
                   I_GeneralPB := #IO_Modes.LMode.SetPBMan,
                   IO_Modes := #IO_Modes,
                   H_HMI := #H_HMITrfInSet,
                   H_TrfIn := #"H_GBChain2W1S-MoviFitFCPN".H_TrfInSet,
                   H_FncSelInHMI := #H_FncSelInHMI,
                   C_TrfInUsed := #C_Config.TrfInSetUsed,
                   O_TrfInCmd => #TrfInSetCmd,
                   O_TrfInRdyRcv => #TrfInSetRdyRcv,
                   O_TrfInInfeedHold => #TrfInfeedHoldSet,
                   O_TrfInArrived => #TrfInSetArrived,
                   O_StopTrfOutCmd => #StopTrfOutSetCmd,
                   O_TrfInActive => #TrfInSetActive,
                   O_TrfInFinished => #TrfInSetFinished,
                   O_InterlockAlarm => #AD_TrfInSetInterlock);
   END_IF;
END_REGION

REGION Network 21: **** 7.1 - Submodule - Non-Machine **** Transfer Out Set
   // Transfer Out Set
   IF "TRUE" THEN
       #_LTrfOutSet(I_StopDet := #I_ExitDet,   // "LGBTrfOut"
                    I_LocalPB := #I_PBSet,
                    I_TrfOutBegin := #I_TrfOutSetBegin,
                    I_TrfOutRdyRcv := #I_TrfOutSetRdyRcv,
                    I_TrfOutInfeedHold := #TrfInfeedHoldSet AND NOT #IO_Modes.LMode.ForcedMan,
                    I_StopTrfOutCmd := "FALSE",
                    I_TrfOutArrived := #I_TrfOutSetArrived,
                    I_ProductionStop := #IO_Modes.LProductionMode.ProdStpMode OR #IO_Modes.LProductionMode.ProdStpModeSel,
                    I_InterlockOk := #I_TrfOutSetIntlkOk,
                    I_ReadyForOperation := #ReadyForOperation,
                    I_SafetyOk := #SafetyOk,
                    I_EnableAlarm := #C_Config.EnableAlarmTransfer,
                    I_ForcedMan := #IO_Modes.LMode.ForcedMan,
                    I_GenRevSw := #IO_Modes.LGeneralFunc.GenRevSwitch,
                    I_GeneralPB := #IO_Modes.LMode.SetPBMan,
                    IO_Modes := #IO_Modes,
                    H_HMI := #H_HMITrfOutSet,
                    H_TrfOut := #"H_GBChain2W1S-MoviFitFCPN".H_TrfOutSet,
                    H_FncSelInHMI := #H_FncSelInHMI,
                    C_TrfMaxTime := #C_Config.TrfMaxTime,
                    C_TrfMaxTimeAfterOvertime := #C_Config.TrfMaxTimeAfterOvertime,
                    C_TrfOutUsed := #C_Config.TrfOutSetUsed,
                    C_EnableTimeoutAlarm := "TRUE",
                    O_TrfOutCmd => #TrfOutSetCmd,
                    O_TrfOutRdyDlv => #TrfOutSetRdyDlv,
                    O_TrfOutOutfeedHold => #TrfOutfeedHoldSet,
                    O_TrfOutTM => #TrfOutSetTM,
                    O_TrfOutActive => #TrfOutSetActive,
                    O_TrfOutFinished => #TrfOutSetFinished,
                    O_OvertimeAlarm => #AC_TrfOutSetOverTime,
                    O_InterlockAlarm => #AD_TrfOutSetInterlock,
                    O_ConfigCalibrationAlm => #AC_ConfigCalibrationAlm,
                    O_CalibrationWarn => #AD_CalibrationSetWarn,
                    O_AlarmABCondition => #TrfOutSetAlmCond);
   END_IF;
END_REGION

REGION Network 22: **** 7.1 - Submodule - Non-Machine **** Transfer IN Set Move UDT
   // Transfer IN Set Move UDT
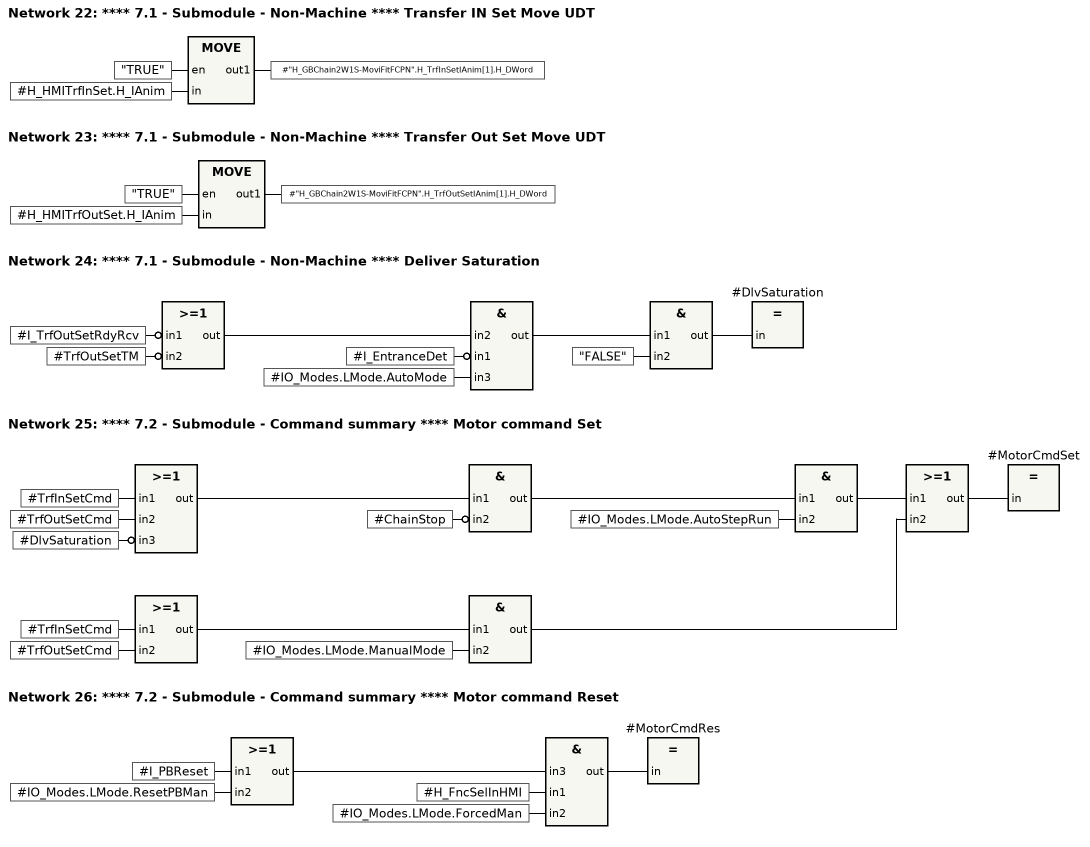
   IF "TRUE" THEN #"H_GBChain2W1S-MoviFitFCPN".H_TrfInSetIAnim[1].H_DWord := #H_HMITrfInSet.H_IAnim; END_IF;
END_REGION

REGION Network 23: **** 7.1 - Submodule - Non-Machine **** Transfer Out Set Move UDT
   // Transfer Out Set Move UDT
   IF "TRUE" THEN
       #"H_GBChain2W1S-MoviFitFCPN".H_TrfOutSetIAnim[1].H_DWord := #H_HMITrfOutSet.H_IAnim;
   END_IF;
END_REGION

REGION Network 24: **** 7.1 - Submodule - Non-Machine **** Deliver Saturation
   #DlvSaturation := (NOT #I_TrfOutSetRdyRcv OR NOT #TrfOutSetTM) AND NOT #I_EntranceDet AND #IO_Modes.LMode.AutoMode AND "FALSE";
END_REGION

REGION Network 25: **** 7.2 - Submodule - Command summary **** Motor command Set
   // Motor command High Speed Set
   #MotorCmdSet := ((#TrfInSetCmd OR #TrfOutSetCmd OR NOT #DlvSaturation) AND NOT #ChainStop AND #IO_Modes.LMode.AutoStepRun) OR ((#TrfInSetCmd OR #TrfOutSetCmd) AND #IO_Modes.LMode.ManualMode);
END_REGION

REGION Network 26: **** 7.2 - Submodule - Command summary **** Motor command Reset
   // Motor command Reset
   #MotorCmdRes := (#I_PBReset OR #IO_Modes.LMode.ResetPBMan) AND #H_FncSelInHMI AND #IO_Modes.LMode.ForcedMan;
END_REGION

REGION Network 27: **** 7.3 - Submodule - Machine **** Motor loop MOVIFIT-FC
   // Motor loop MOVIFIT-FC
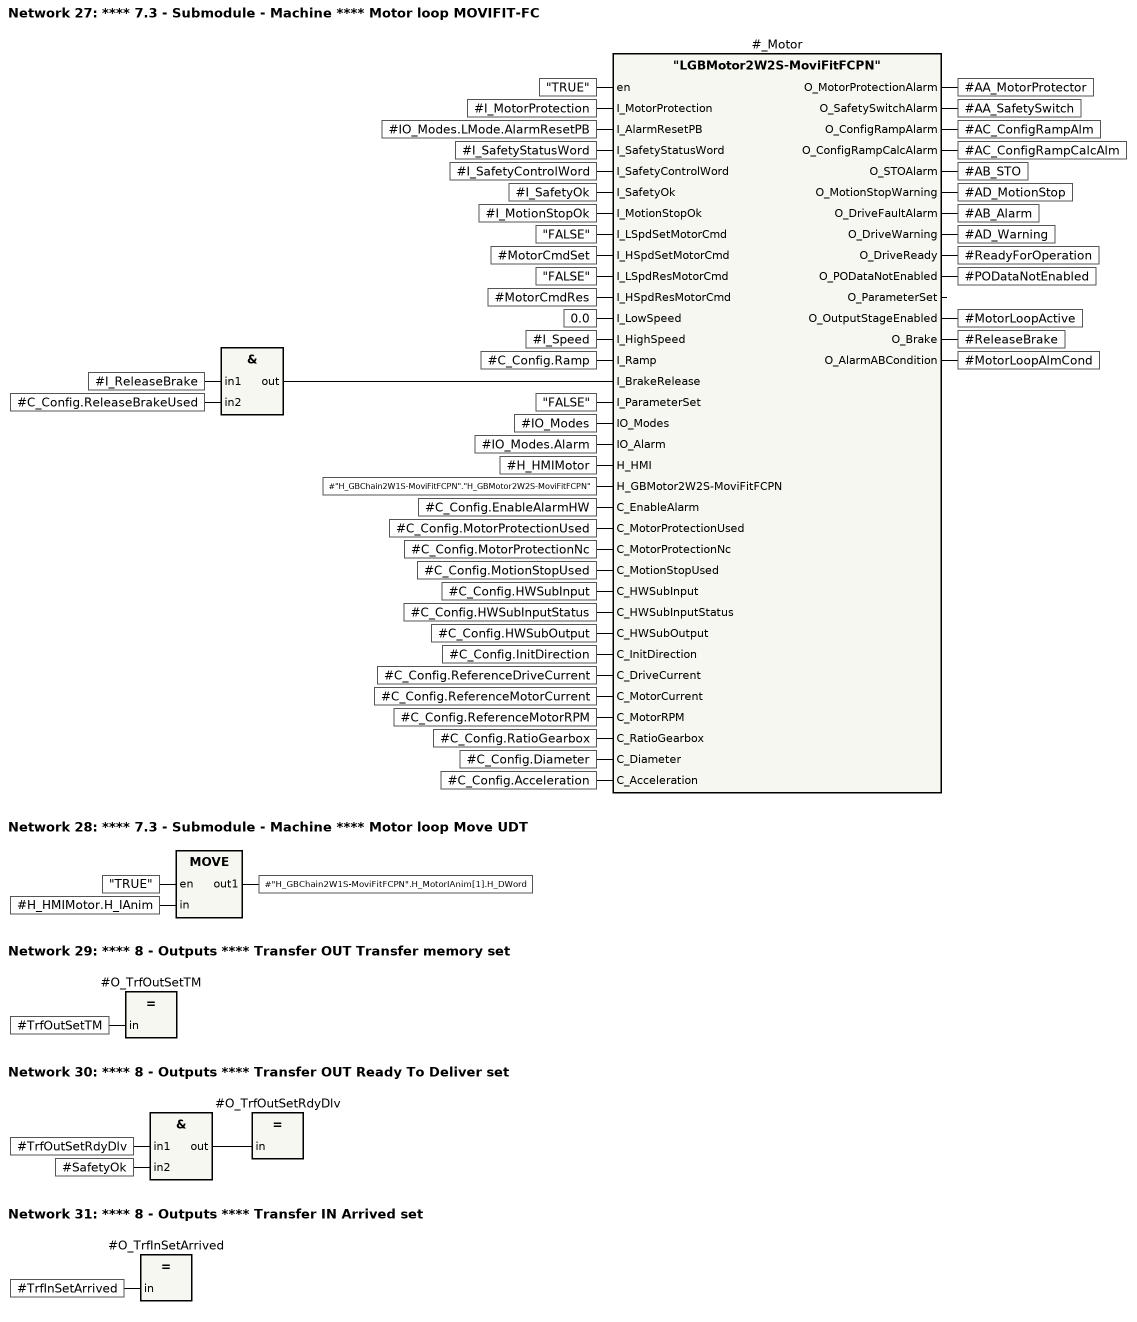
   IF "TRUE" THEN
       #_Motor(I_MotorProtection := #I_MotorProtection,   // "LGBMotor2W2S-MoviFitFCPN"
               I_AlarmResetPB := #IO_Modes.LMode.AlarmResetPB,
               I_SafetyStatusWord := #I_SafetyStatusWord,
               I_SafetyControlWord := #I_SafetyControlWord,
               I_SafetyOk := #I_SafetyOk,
               I_MotionStopOk := #I_MotionStopOk,
               I_LSpdSetMotorCmd := "FALSE",
               I_HSpdSetMotorCmd := #MotorCmdSet,
               I_LSpdResMotorCmd := "FALSE",
               I_HSpdResMotorCmd := #MotorCmdRes,
               I_LowSpeed := 0.0,
               I_HighSpeed := #I_Speed,
               I_Ramp := #C_Config.Ramp,
               I_BrakeRelease := #I_ReleaseBrake AND #C_Config.ReleaseBrakeUsed,
               I_ParameterSet := "FALSE",
               IO_Modes := #IO_Modes,
               IO_Alarm := #IO_Modes.Alarm,
               H_HMI := #H_HMIMotor,
               "H_GBMotor2W2S-MoviFitFCPN" := #"H_GBChain2W1S-MoviFitFCPN"."H_GBMotor2W2S-MoviFitFCPN",
               C_EnableAlarm := #C_Config.EnableAlarmHW,
               C_MotorProtectionUsed := #C_Config.MotorProtectionUsed,
               C_MotorProtectionNc := #C_Config.MotorProtectionNc,
               C_MotionStopUsed := #C_Config.MotionStopUsed,
               C_HWSubInput := #C_Config.HWSubInput,
               C_HWSubInputStatus := #C_Config.HWSubInputStatus,
               C_HWSubOutput := #C_Config.HWSubOutput,
               C_InitDirection := #C_Config.InitDirection,
               C_DriveCurrent := #C_Config.ReferenceDriveCurrent,
               C_MotorCurrent := #C_Config.ReferenceMotorCurrent,
               C_MotorRPM := #C_Config.ReferenceMotorRPM,
               C_RatioGearbox := #C_Config.RatioGearbox,
               C_Diameter := #C_Config.Diameter,
               C_Acceleration := #C_Config.Acceleration,
               O_MotorProtectionAlarm => #AA_MotorProtector,
               O_SafetySwitchAlarm => #AA_SafetySwitch,
               O_ConfigRampAlarm => #AC_ConfigRampAlm,
               O_ConfigRampCalcAlarm => #AC_ConfigRampCalcAlm,
               O_STOAlarm => #AB_STO,
               O_MotionStopWarning => #AD_MotionStop,
               O_DriveFaultAlarm => #AB_Alarm,
               O_DriveWarning => #AD_Warning,
               O_DriveReady => #ReadyForOperation,
               O_PODataNotEnabled => #PODataNotEnabled,
               O_OutputStageEnabled => #MotorLoopActive,
               O_Brake => #ReleaseBrake,
               O_AlarmABCondition => #MotorLoopAlmCond);
   END_IF;
END_REGION

REGION Network 28: **** 7.3 - Submodule - Machine **** Motor loop Move UDT
   IF "TRUE" THEN #"H_GBChain2W1S-MoviFitFCPN".H_MotorIAnim[1].H_DWord := #H_HMIMotor.H_IAnim; END_IF;
END_REGION

REGION Network 29: **** 8 - Outputs **** Transfer OUT Transfer memory set
   // Transfer OUT Transfer memory set
   #O_TrfOutSetTM := #TrfOutSetTM;
END_REGION

REGION Network 30: **** 8 - Outputs **** Transfer OUT Ready To Deliver set
   // Transfer OUT Ready To Deliver set
   #O_TrfOutSetRdyDlv := #TrfOutSetRdyDlv AND #SafetyOk;
END_REGION

REGION Network 31: **** 8 - Outputs **** Transfer IN Arrived set
   // Transfer IN Arrived set
   #O_TrfInSetArrived := #TrfInSetArrived;
END_REGION

REGION Network 32: **** 8 - Outputs **** Transfer IN Ready To Receive set
   // Transfer IN Ready To Receive set
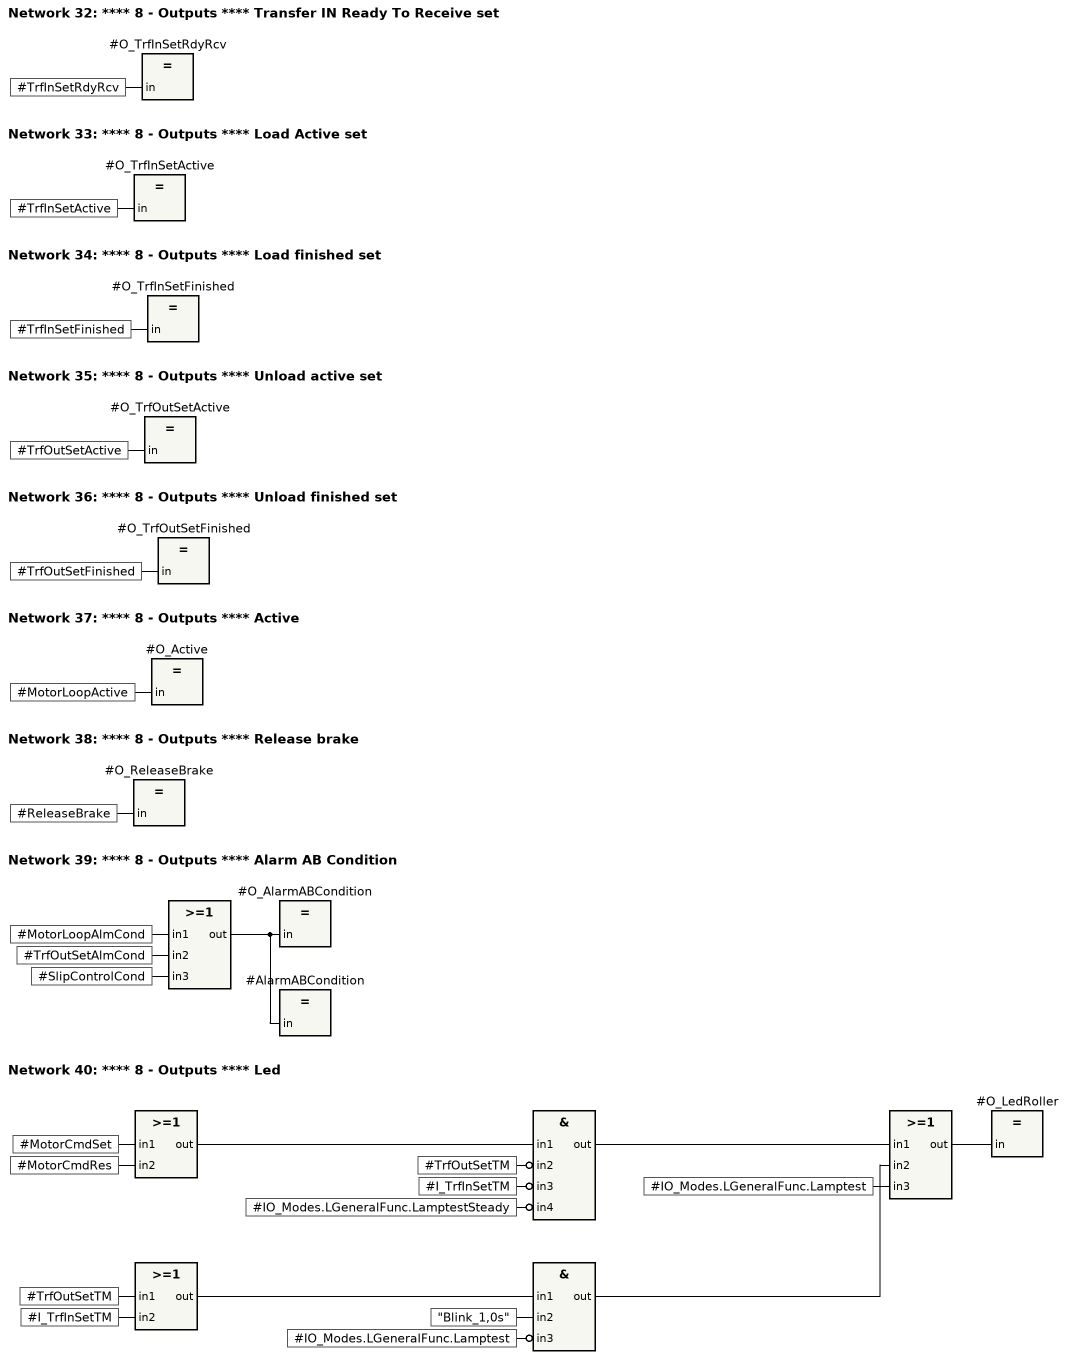
   #O_TrfInSetRdyRcv := #TrfInSetRdyRcv;
END_REGION

REGION Network 33: **** 8 - Outputs **** Load Active set
   // Load Active set
   #O_TrfInSetActive := #TrfInSetActive;
END_REGION

REGION Network 34: **** 8 - Outputs **** Load finished set
   // Load finished set
   #O_TrfInSetFinished := #TrfInSetFinished;
END_REGION

REGION Network 35: **** 8 - Outputs **** Unload active set
   // Unload active set
   #O_TrfOutSetActive := #TrfOutSetActive;
END_REGION

REGION Network 36: **** 8 - Outputs **** Unload finished set
   // Unload finished set
   #O_TrfOutSetFinished := #TrfOutSetFinished;
END_REGION

REGION Network 37: **** 8 - Outputs **** Active
   // Active
   #O_Active := #MotorLoopActive;
END_REGION

REGION Network 38: **** 8 - Outputs **** Release brake
   // Release brake
   #O_ReleaseBrake := #ReleaseBrake;
END_REGION

REGION Network 39: **** 8 - Outputs **** Alarm AB Condition
   // Alarm AB Condition
   #O_AlarmABCondition := #MotorLoopAlmCond OR #TrfOutSetAlmCond OR #SlipControlCond;
   #AlarmABCondition := #O_AlarmABCondition;
END_REGION

REGION Network 40: **** 8 - Outputs **** Led
   // Led
   #O_LedRoller := ((#MotorCmdSet OR #MotorCmdRes) AND NOT #TrfOutSetTM AND NOT #I_TrfInSetTM AND NOT #IO_Modes.LGeneralFunc.LamptestSteady) OR ((#TrfOutSetTM OR #I_TrfInSetTM) AND "Blink_1,0s" AND NOT #IO_Modes.LGeneralFunc.Lamptest) OR #IO_Modes.LGeneralFunc.Lamptest;
END_REGION

REGION Network 41: **** 8 - Outputs **** Occupied
   // Occupied
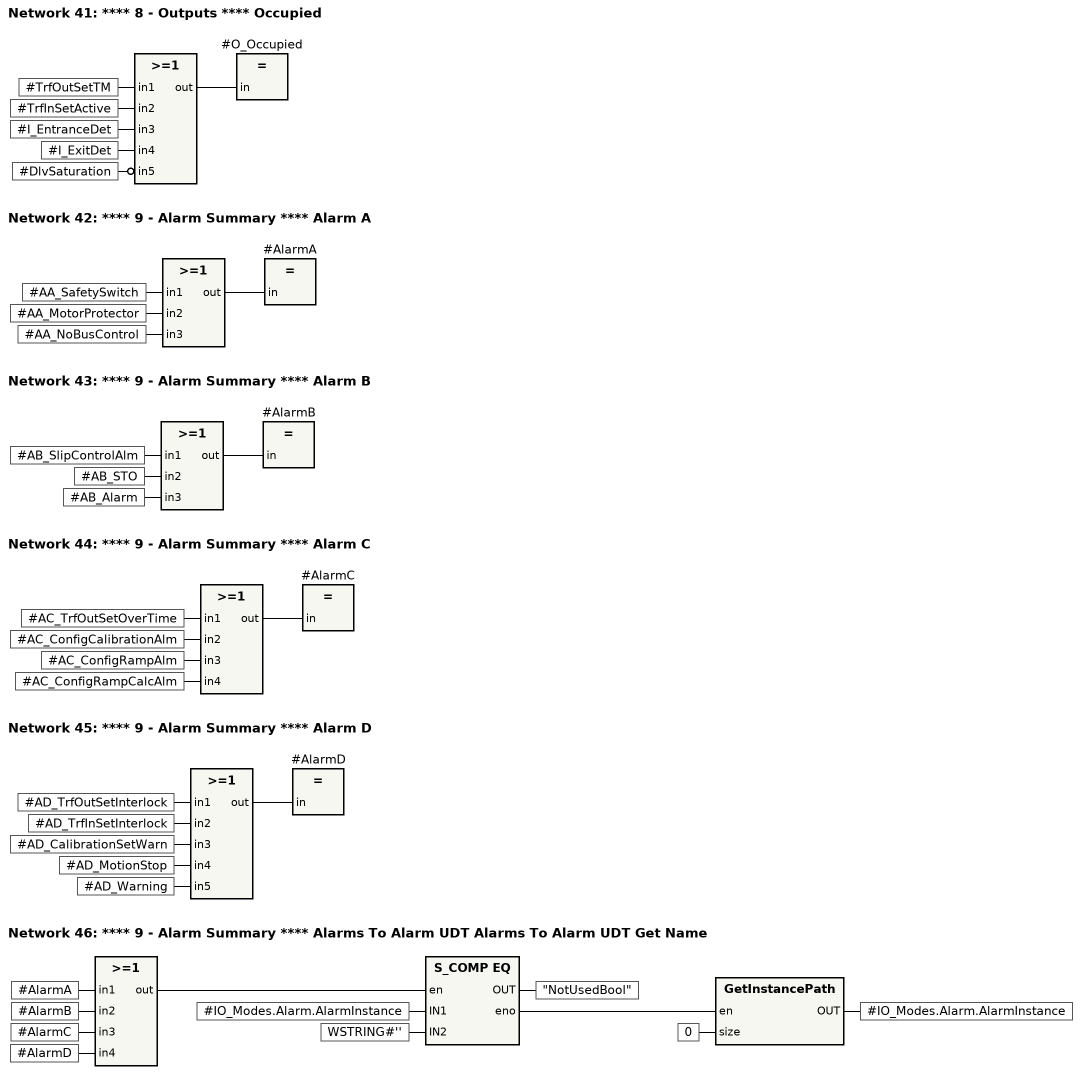
   #O_Occupied := #TrfOutSetTM OR #TrfInSetActive OR #I_EntranceDet OR #I_ExitDet OR NOT #DlvSaturation;
END_REGION

REGION Network 42: **** 9 - Alarm Summary **** Alarm A
   // Alarm A
   #AlarmA := #AA_SafetySwitch OR #AA_MotorProtector OR #AA_NoBusControl;
END_REGION

REGION Network 43: **** 9 - Alarm Summary **** Alarm B
   // Alarm B
   #AlarmB := #AB_SlipControlAlm OR #AB_STO OR #AB_Alarm;
END_REGION

REGION Network 44: **** 9 - Alarm Summary **** Alarm C
   // Alarm C
   #AlarmC := #AC_TrfOutSetOverTime OR #AC_ConfigCalibrationAlm OR #AC_ConfigRampAlm OR #AC_ConfigRampCalcAlm;
END_REGION

REGION Network 45: **** 9 - Alarm Summary **** Alarm D
   // Alarm D
   #AlarmD := #AD_TrfOutSetInterlock OR #AD_TrfInSetInterlock OR #AD_CalibrationSetWarn OR #AD_MotionStop OR #AD_Warning;
END_REGION

REGION Network 46: **** 9 - Alarm Summary **** Alarms To Alarm UDT Alarms To Alarm UDT Get Name
   // Alarm D
   S_COMP(EN := #AlarmA OR #AlarmB OR #AlarmC OR #AlarmD,
          IN1 := #IO_Modes.Alarm.AlarmInstance,
          IN2 := WSTRING#'',
          OUT => "NotUsedBool",
          ENO => #_w1);
   IF #_w1 THEN GetInstancePath(size := 0, OUT => #IO_Modes.Alarm.AlarmInstance); END_IF;
END_REGION

REGION Network 47: **** 9 - Alarm Summary **** Alarms To Alarm UDT
   // Alarm D
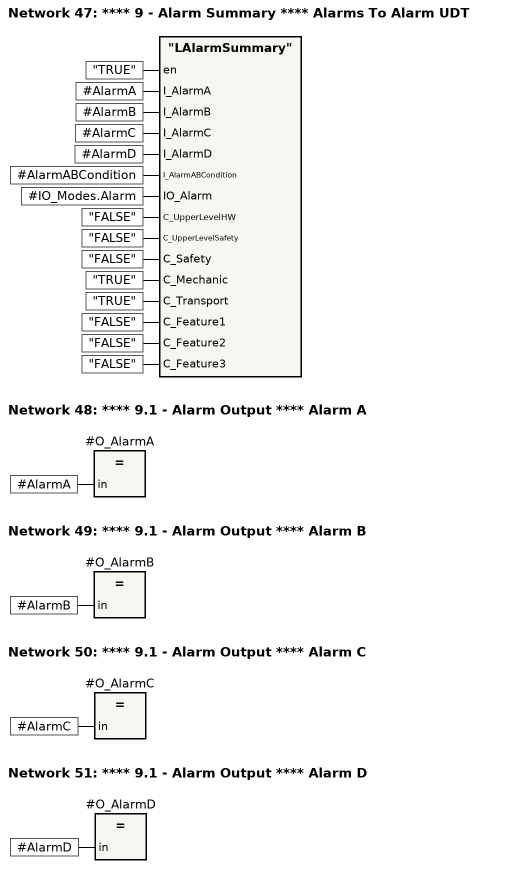
   IF "TRUE" THEN
       "LAlarmSummary"(I_AlarmA := #AlarmA,
                       I_AlarmB := #AlarmB,
                       I_AlarmC := #AlarmC,
                       I_AlarmD := #AlarmD,
                       I_AlarmABCondition := #AlarmABCondition,
                       IO_Alarm := #IO_Modes.Alarm,
                       C_UpperLevelHW := "FALSE",
                       C_UpperLevelSafety := "FALSE",
                       C_Safety := "FALSE",
                       C_Mechanic := "TRUE",
                       C_Transport := "TRUE",
                       C_Feature1 := "FALSE",
                       C_Feature2 := "FALSE",
                       C_Feature3 := "FALSE");
   END_IF;
END_REGION

REGION Network 48: **** 9.1 - Alarm Output **** Alarm A
   // Alarm A
   #O_AlarmA := #AlarmA;
END_REGION

REGION Network 49: **** 9.1 - Alarm Output **** Alarm B
   // Alarm B
   #O_AlarmB := #AlarmB;
END_REGION

REGION Network 50: **** 9.1 - Alarm Output **** Alarm C
   // Alarm C
   #O_AlarmC := #AlarmC;
END_REGION

REGION Network 51: **** 9.1 - Alarm Output **** Alarm D
   // Alarm D
   #O_AlarmD := #AlarmD;
END_REGION

REGION Network 52: **** 9.2 - Alarm DWord**** Alarm To DWord
   // Alarm Word
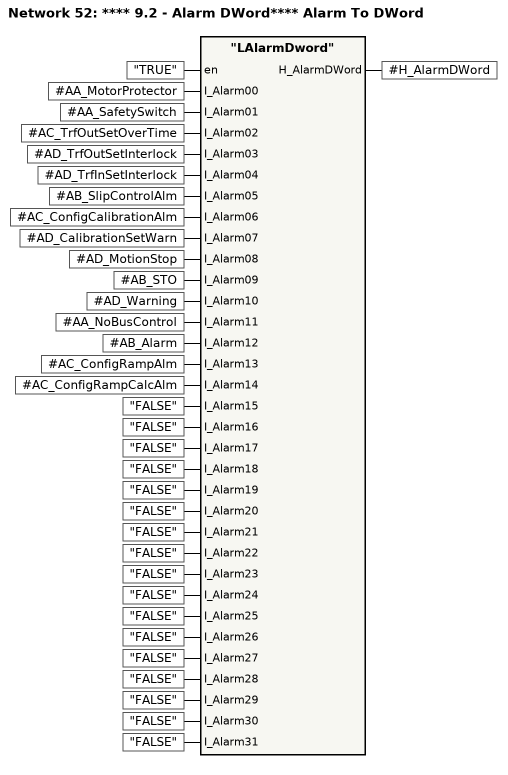
   IF "TRUE" THEN
       "LAlarmDword"(I_Alarm00 := #AA_MotorProtector,
                     I_Alarm01 := #AA_SafetySwitch,
                     I_Alarm02 := #AC_TrfOutSetOverTime,
                     I_Alarm03 := #AD_TrfOutSetInterlock,
                     I_Alarm04 := #AD_TrfInSetInterlock,
                     I_Alarm05 := #AB_SlipControlAlm,
                     I_Alarm06 := #AC_ConfigCalibrationAlm,
                     I_Alarm07 := #AD_CalibrationSetWarn,
                     I_Alarm08 := #AD_MotionStop,
                     I_Alarm09 := #AB_STO,
                     I_Alarm10 := #AD_Warning,
                     I_Alarm11 := #AA_NoBusControl,
                     I_Alarm12 := #AB_Alarm,
                     I_Alarm13 := #AC_ConfigRampAlm,
                     I_Alarm14 := #AC_ConfigRampCalcAlm,
                     I_Alarm15 := "FALSE",
                     I_Alarm16 := "FALSE",
                     I_Alarm17 := "FALSE",
                     I_Alarm18 := "FALSE",
                     I_Alarm19 := "FALSE",
                     I_Alarm20 := "FALSE",
                     I_Alarm21 := "FALSE",
                     I_Alarm22 := "FALSE",
                     I_Alarm23 := "FALSE",
                     I_Alarm24 := "FALSE",
                     I_Alarm25 := "FALSE",
                     I_Alarm26 := "FALSE",
                     I_Alarm27 := "FALSE",
                     I_Alarm28 := "FALSE",
                     I_Alarm29 := "FALSE",
                     I_Alarm30 := "FALSE",
                     I_Alarm31 := "FALSE",
                     H_AlarmDWord => #H_AlarmDWord);
   END_IF;
END_REGION
END_FUNCTION_BLOCK
